# B&R Automation Studio project OpcUaSample410_BrbLibUa103 (part 21)

#### Action.st
```iecst
ACTION InitAirCond:
	// Logik
	pInstance.Act.eOperationMode := eAC_OPERATIONMODE_OFF;
	pInstance.Act.rTemperature := rAIR_COND_TEMP_OUTSIDE;
	pInstance.Act.nFanLevel := 0;
	pInstance.Set.rTemperature := 20.0;
	pInstance.Set.nFanLevel := 0;
END_ACTION

ACTION OperateAirCond:
	// Methode 'SetOperationMode'
	CASE pIntern.MethSetOperationMode.nStep OF
		0:
			// Prüfen, ob Methode von einem Client aufgerufen wurde
			pIntern.MethSetOperationMode.fbUaSrv_MethodOperate.Execute := 1;
			pIntern.MethSetOperationMode.fbUaSrv_MethodOperate.Action := UaMoa_CheckIsCalled;
			IF pIntern.MethSetOperationMode.fbUaSrv_MethodOperate.Done = 1 THEN
				pIntern.MethSetOperationMode.fbUaSrv_MethodOperate.Execute := 0;
				IF pIntern.MethSetOperationMode.fbUaSrv_MethodOperate.IsCalled = 1 THEN
					// Variablen der Eingans-Argumente sind besetzt -> Methode ausführen
					pIntern.MethSetOperationMode.nStep := 1;
				END_IF
			ELSIF pIntern.MethSetOperationMode.fbUaSrv_MethodOperate.Error = 1 THEN
				// Fehler, aber trotzdem weiter machen
				pIntern.MethSetOperationMode.fbUaSrv_MethodOperate.Execute := 0;
			END_IF

		1:
			// Ausführen der Methode
			IF pIntern.MethSetOperationMode.ArgsIn.eOperationMode >= eAC_OPERATIONMODE_OFF AND pIntern.MethSetOperationMode.ArgsIn.eOperationMode <= eAC_OPERATIONMODE_AUTO THEN
				pInstance.Act.eOperationMode := pIntern.MethSetOperationMode.ArgsIn.eOperationMode;
				pIntern.MethSetOperationMode.ArgsOut.eStatus := eAC_METH_STATUS_OK;
			ELSE
				pIntern.MethSetOperationMode.ArgsOut.eStatus := eAC_METH_STATUS_INVALID_OPMODE;
			END_IF
			pIntern.MethSetOperationMode.nStep := 2;

		2:
			// Rückmelden, dass Methode ausgeführt wurde. Zu diesem Zeitpunkt müssen die Ausgangs-Argumente besetzt sein und dürfen nicht mehr geändert werden
			pIntern.MethSetOperationMode.fbUaSrv_MethodOperate.Execute := 1;
			pIntern.MethSetOperationMode.fbUaSrv_MethodOperate.Action := UaMoa_Finished;
			IF pIntern.MethSetOperationMode.fbUaSrv_MethodOperate.Done = 1 THEN
				pIntern.MethSetOperationMode.fbUaSrv_MethodOperate.Execute := 0;
				pIntern.MethSetOperationMode.nStep := 0;
			ELSIF pIntern.MethSetOperationMode.fbUaSrv_MethodOperate.Error = 1 THEN
				// Fehler, aber trotzdem weiter machen
				pIntern.MethSetOperationMode.fbUaSrv_MethodOperate.Execute := 0;
				pIntern.MethSetOperationMode.nStep := 0;
			END_IF

	END_CASE
	pIntern.MethSetOperationMode.fbUaSrv_MethodOperate();

	// Begrenzung der SetTemp
	IF pInstance.Set.rTemperature < rAIR_COND_TEMP_MIN THEN
		pInstance.Set.rTemperature := rAIR_COND_TEMP_MIN;
	ELSIF pInstance.Set.rTemperature > rAIR_COND_TEMP_OUTSIDE THEN
		pInstance.Set.rTemperature := rAIR_COND_TEMP_OUTSIDE;
	END_IF
	// Berechnung der internen Werte (Abweichung in Prozent)
	pIntern.rDiff := pInstance.Act.rTemperature - pInstance.Set.rTemperature;
	pIntern.rDiffPercent := pIntern.rDiff / pInstance.Act.rTemperature * 100.0;
	// Steuern des Lüfters
	IF pInstance.Act.eOperationMode = eAC_OPERATIONMODE_OFF THEN
		// Lüfter ausschalten
		pInstance.Act.nFanLevel := 0;
	ELSIF pInstance.Act.eOperationMode = eAC_OPERATIONMODE_MANUAL THEN
		// Lüfter-Stufe aus manueller Vorgabe übernehmen
		IF pInstance.Set.nFanLevel > 5 THEN
			pInstance.Act.nFanLevel := 5;
		ELSE
			pInstance.Act.nFanLevel := pInstance.Set.nFanLevel;
		END_IF
	ELSIF pInstance.Act.eOperationMode = eAC_OPERATIONMODE_AUTO THEN
		// Lüfter-Stufe je nach Temperatur-Differenz setzen
		IF pIntern.rDiffPercent <= 0.0 THEN
			pInstance.Act.nFanLevel := 0;
		ELSIF pIntern.rDiffPercent <= 10.0 THEN
			pInstance.Act.nFanLevel := 1;
		ELSIF pIntern.rDiffPercent <= 15.0 THEN
			pInstance.Act.nFanLevel := 2;
		ELSIF pIntern.rDiffPercent <= 20.0 THEN
			pInstance.Act.nFanLevel := 3;
		ELSIF pIntern.rDiffPercent <= 25.0 THEN
			pInstance.Act.nFanLevel := 4;
		ELSE
			pInstance.Act.nFanLevel := 5;
		END_IF
	END_IF
	SimulateAirCond;

	// Event 'AirConditionOperationModeChanged'
	IF pInstance.Act.eOperationMode <> pIntern.EvntOperationModeChanged.eOldOperationMode THEN
		// Besetzen der Felder mit aktuellen Werten
		pIntern.EvntOperationModeChanged.Fields.OldOperationMode := pIntern.EvntOperationModeChanged.eOldOperationMode;
		pIntern.EvntOperationModeChanged.Fields.NewOperationMode := pInstance.Act.eOperationMode;
		sMessageText := 'Operation mode of air condition $'';
		brsstrcat(ADR(sMessageText), ADR(pInstance.sName));
		brsstrcat(ADR(sMessageText), ADR('$' has changed from $''));
		eOperationMode := pIntern.EvntOperationModeChanged.Fields.OldOperationMode;
		GetOperationModeText;
		brsstrcat(ADR(sMessageText), ADR(sOperationModeText));
		brsstrcat(ADR(sMessageText), ADR('$' to $''));
		eOperationMode := pIntern.EvntOperationModeChanged.Fields.NewOperationMode;
		GetOperationModeText;
		brsstrcat(ADR(sMessageText), ADR(sOperationModeText));
		brsstrcat(ADR(sMessageText), ADR('$' (ST).'));
		brsstrcpy(ADR(pIntern.EvntOperationModeChanged.Fields.Message.Text), ADR(sMessageText));
		// Event feuern
		pIntern.EvntOperationModeChanged.bFire := 1;
	END_IF
	pIntern.EvntOperationModeChanged.eOldOperationMode := pInstance.Act.eOperationMode;
	CASE pIntern.EvntOperationModeChanged.nStep OF
		0:
			// Ermitteln des Namespace-Index für Fremdmodell-Adressbereich am am B&R-Server
			pIntern.EvntOperationModeChanged.fbUaSrv_GetNamespaceIndex.Execute := 1;
			pIntern.EvntOperationModeChanged.fbUaSrv_GetNamespaceIndex.NamespaceUri := 'http://br-automation.com/AirCondModel/';
			IF pIntern.EvntOperationModeChanged.fbUaSrv_GetNamespaceIndex.Done = 1 THEN
				pIntern.EvntOperationModeChanged.fbUaSrv_GetNamespaceIndex.Execute := 0;
				pIntern.EvntOperationModeChanged.nNamespaceIndexAirCond := pIntern.EvntOperationModeChanged.fbUaSrv_GetNamespaceIndex.NamespaceIndex;
				brsitoa(pIntern.EvntOperationModeChanged.nNamespaceIndexAirCond, ADR(pIntern.EvntOperationModeChanged.sNamespaceIndexAirCond));
				pIntern.EvntOperationModeChanged.nStep := pIntern.EvntOperationModeChanged.nStep + 1;
			ELSIF pIntern.EvntOperationModeChanged.fbUaSrv_GetNamespaceIndex.Error = 1 THEN
				// Fehler
				pIntern.EvntOperationModeChanged.fbUaSrv_GetNamespaceIndex.Execute := 0;
			END_IF

		1:
			// Initialisierung zum Feuern des Events
			// Event-Typ
			pIntern.EvntOperationModeChanged.fbUaSrv_FireEvent.EventType.NamespaceIndex := pIntern.EvntOperationModeChanged.nNamespaceIndexAirCond;
			pIntern.EvntOperationModeChanged.fbUaSrv_FireEvent.EventType.IdentifierType := UAIdentifierType_Numeric;
			pIntern.EvntOperationModeChanged.fbUaSrv_FireEvent.EventType.Identifier := '1002'; // = AirConditionOperationModeChanged
			// Event-Felder
			nFieldIndex := 0;
			// SourceNode
			pIntern.EvntOperationModeChanged.Fields.FieldCfg[nFieldIndex].BrowsePath := '/SourceNode';
			sVarNameTotal := pIntern.EvntOperationModeChanged.sEventFieldsBaseVarName;
			brsstrcat(ADR(sVarNameTotal), ADR('.SourceNode'));
			pIntern.EvntOperationModeChanged.Fields.FieldCfg[nFieldIndex].Variable := sVarNameTotal;
			pIntern.EvntOperationModeChanged.Fields.SourceNode.NamespaceIndex := pIntern.EvntOperationModeChanged.nNamespaceIndexAirCond;
			pIntern.EvntOperationModeChanged.Fields.SourceNode.IdentifierType := UAIdentifierType_Numeric;
			pIntern.EvntOperationModeChanged.Fields.SourceNode.Identifier := pIntern.EvntOperationModeChanged.sEventFieldSourceNode;
			// Message
			nFieldIndex := nFieldIndex + 1;
			pIntern.EvntOperationModeChanged.Fields.FieldCfg[nFieldIndex].BrowsePath := '/Message';
			sVarNameTotal := pIntern.EvntOperationModeChanged.sEventFieldsBaseVarName;
			brsstrcat(ADR(sVarNameTotal), ADR('.Message'));
			pIntern.EvntOperationModeChanged.Fields.FieldCfg[nFieldIndex].Variable := sVarNameTotal;
			pIntern.EvntOperationModeChanged.Fields.Message.Text := 'Operation mode has changed.';
			// OldOperationMode
			nFieldIndex := nFieldIndex + 1;
			sFieldNameTotal := '/';
			brsstrcat(ADR(sFieldNameTotal), ADR(pIntern.EvntOperationModeChanged.sNamespaceIndexAirCond));
			brsstrcat(ADR(sFieldNameTotal), ADR(':OldOperationMode'));
			pIntern.EvntOperationModeChanged.Fields.FieldCfg[nFieldIndex].BrowsePath := sFieldNameTotal;
			sVarNameTotal := pIntern.EvntOperationModeChanged.sEventFieldsBaseVarName;
			brsstrcat(ADR(sVarNameTotal), ADR('.OldOperationMode'));
			pIntern.EvntOperationModeChanged.Fields.FieldCfg[nFieldIndex].Variable := sVarNameTotal;
			// NewOperationMode
			nFieldIndex := nFieldIndex + 1;
			sFieldNameTotal := '/';
			brsstrcat(ADR(sFieldNameTotal), ADR(pIntern.EvntOperationModeChanged.sNamespaceIndexAirCond));
			brsstrcat(ADR(sFieldNameTotal), ADR(':NewOperationMode'));
			pIntern.EvntOperationModeChanged.Fields.FieldCfg[nFieldIndex].BrowsePath := sFieldNameTotal;
			sVarNameTotal := pIntern.EvntOperationModeChanged.sEventFieldsBaseVarName;
			brsstrcat(ADR(sVarNameTotal), ADR('.NewOperationMode'));
			pIntern.EvntOperationModeChanged.Fields.FieldCfg[nFieldIndex].Variable := sVarNameTotal;
			// Statische Funktionsblock-Eingänge
			pIntern.EvntOperationModeChanged.fbUaSrv_FireEvent.EventFieldCount := nFieldIndex+1;
			pIntern.EvntOperationModeChanged.nStep := pIntern.EvntOperationModeChanged.nStep + 1;

		2:
			// Prüfen, ob Event gefeuert werden muss
			IF pIntern.EvntOperationModeChanged.bFire = 1 THEN
				pIntern.EvntOperationModeChanged.bFire := 0;
				pIntern.EvntOperationModeChanged.nStep := pIntern.EvntOperationModeChanged.nStep + 1;
			END_IF

		3:
			// Event feuern
			pIntern.EvntOperationModeChanged.fbUaSrv_FireEvent.Execute := 1;
			IF pIntern.EvntOperationModeChanged.fbUaSrv_FireEvent.Done = 1 THEN
				pIntern.EvntOperationModeChanged.fbUaSrv_FireEvent.Execute := 0;
				pIntern.EvntOperationModeChanged.nStep := pIntern.EvntOperationModeChanged.nStep - 1;
			ELSIF pIntern.EvntOperationModeChanged.fbUaSrv_FireEvent.Error = 1 THEN
				// Fehler
			END_IF

	END_CASE
	pIntern.EvntOperationModeChanged.fbUaSrv_GetNamespaceIndex();
	pIntern.EvntOperationModeChanged.fbUaSrv_FireEvent(EventFields := pIntern.EvntOperationModeChanged.Fields.FieldCfg[0]);

END_ACTION

ACTION SimulateAirCond:
	// Stetiges Angleichen an die Aussentemperatur
	pInstance.Act.rTemperature := pInstance.Act.rTemperature + 0.0005;
	IF pInstance.Act.rTemperature > rAIR_COND_TEMP_OUTSIDE THEN
		pInstance.Act.rTemperature := rAIR_COND_TEMP_OUTSIDE;
	END_IF
	// Kühlen
	IF pInstance.Act.eOperationMode <> eAC_OPERATIONMODE_OFF THEN
		// Je nach Lüfter-Stufe kühlt die ActTemp runter
		pIntern.rCoolStepTemp := pInstance.Act.nFanLevel * 0.005;
		pInstance.Act.rTemperature := pInstance.Act.rTemperature - pIntern.rCoolStepTemp;
	END_IF
	// Physikalische Begrenzung der ActTemp
	IF pInstance.Act.rTemperature < rAIR_COND_TEMP_MIN THEN
		pInstance.Act.rTemperature := rAIR_COND_TEMP_MIN;
	END_IF
END_ACTION

ACTION GetOperationModeText:
	IF eOperationMode = eAC_OPERATIONMODE_OFF THEN
		sOperationModeText := 'Off';
	ELSIF eOperationMode = eAC_OPERATIONMODE_MANUAL THEN
		sOperationModeText := 'Manual';
	ELSIF eOperationMode = eAC_OPERATIONMODE_AUTO THEN
		sOperationModeText := 'Automatic';
	ELSE
		sOperationModeText := 'Unknown';
	END_IF
END_ACTION
```

### ReadMe.txt
```
Hier wird die Konfiguration von Publisher/Subscriber gezeigt.

Allgemeines zu PubSub
	PubSub ist eine alternative OpcUa-Kommunikation zu einer Client-Server-Verbindung.
	Bei PubSub ist es im Gegensatz zu Client/Server nicht notwendig, eine explizite Verbindung aufzubauen. Der Publisher
	schickt die Daten autark durch ein Udp-Multicast-Telegramm ins Netzwerk. Dieses	Telegramm kann dann von einem oder
	mehreren Subscribern empfangen und ausgewertet werden. Der Publisher weiss nicht, ob und welche Subscriber zuhören.
	Eine B&R-Sps kann Publisher sein (und mehrere Datenblöcke in verschiedenen Intervallen publishen) und gleichzeitig
	Subscriber auf mehrere andere Publisher enthalten. Sie kann sich nur nicht auf einen Datenblock des eigenen Publishers
	abonnieren (Hintergrund siehe 'Zu diesem Beispiel' unten).

	Theoretisch muss ein Publisher oder ein Subscriber nicht gleichzeitig ein Server oder Client sein. Beide Kommunkationsarten
	haben lt. Spezifikation nichts miteinander zu tun.
	Praktisch ist es aber oft so, dass ein Publisher Knoten aus einem Adressraum veröffentlicht, der bequemerweise von einem
	Server bereitgestellt wird. Auch ein Subscriber benötigt einen Adressraum, auf dessen Knoten die empfangenen Daten kopiert
	werden können. Eine B&R-Sps braucht deshalb eine Adressraum-Konfiguration und auch das OpcUa-System muss in der System-
	Konfiguration aktiviert sein.

	PubSub wird oft zusammen mit TSN (TimeSensitiveNetwork, also echtzeitfähiges Ethernet) genannt. Tatsächlich wird PubSub
	von OpcUa-TSN verwendet. Trotzdem kann PubSub auch autaurk in nicht echtzeitfähigen Ethernet-Netzwerken eingesetzt
	werden. Dies ist hier der Fall, da TSN noch nicht veröffentlicht ist. Deshalb müssen auch die Parameter unter 'Activate VLAN'
	in der PubSub-Konfiguration noch nicht gesetzt werden (sie sind später für TSN wichtig).

	Laut Spezifikation hängt der Aufbau eines Publisher-Multicast-Telegramms (einer sogenannten NetworkMessage) von sehr
	vielen Optionen ab. Viele Parameter	werden nur optional im Telegramm mitgesendet. Es gibt auch einige spezifizierte
	Formate, sogenannte 'HeaderLayouts', welche den Aufbau zu großen Teilen festlegen. So kann die sonst sehr aufwändige
	Konfiguration stark vereinfacht	ausfallen. B&R nutzt das HeaderLayout 'UADP-Periodic-Fixed', mit dem viele Parameter
	fix gesetzt sind und so die	Konfiguration überschaubar macht.
	Es gibt auch einige Einschränkungen, welche in der AS-Hilfe genauer beschrieben sind:
		-Nur skalare Werte und 1-dimensionale Arrays
		-Keine Strukturen, Enumerationen, Pointer, Konstanten
		-Noch keine Security (Verschlüsselung)
		-Der Publisher wird nicht synchron zu den Taskklassen ausgeführt. Somit ist eine Konsistenz der Daten zueinander, auch
			wenn sie in einem DataSet sind, nicht gewährleistet. Diese Funktionalität wird erst durch TSN abgebildet werden
			können.

Zu diesem Beispiel
	Leider kann in einer ArSim (Sps-Simulation auf einem PC), wie sie für dieses Beispiel-Projekt verwendet wird, keine
	funktionierende PubSub-Verbindung gezeigt werden. Dafür gibt es mehrere Gründe:
		1. Eine Sps kann sich nicht selber zuhören, also auf den eigenen Publisher subscriben.
				Grund: Ethernet-Sockets sind auf der Sps so eingestellt, dass sie ihre gesendeteten Telegramme nicht gleichzeitig
				auch empfangen (auch nicht, wenn es Multicast-Telegramme sind). Dies hat performance-technische Gründe:
				Müsste ein Socket auch die selber gesendeten Telegramme empfangen und auswerten, würde dies die Hardware zu sehr
				durch Interrupts belasten.
		2. Eine ArSim hat normalerweise (wie hier auch) eine virtuelle Ethernet-Verbindung über die Adresse 127.0.0.1.
				Aufgrund des virtuellen Netzwerkes werden keine Telegramme vom Publisher veröffentlicht.

	Aus diesem Grund kann hier nur die exemplarische Konfiguration gezeigt werden. Würde dieses Beispiel auf zwei Hardware-
	Sps angepasst, so würde die Kommunikation funktionieren.

	Es gibt zumindest einen Trick, wie die Publisher-Multicast-Telegramme einer ArSim in ein äußeres Netzwerk des PC's gebracht
	werden können: Die Ip-Adresse der einzigen ArSim-Ethernet-Schnittstelle IF3, welche normalerweise auf 127.0.0.1 eingestellt
	ist, muss auf die Ip-Adresse des PC's zu dem Netzwerk eingestellt werden. Dann werden die Telegramme über Windows automatisch
	an diese Ethernet-Schnittstelle und somit in das Netzwerk geschickt. Sie können dann sogar mit Wireshark aufgezeichnet
	oder von einem Subscriber im Netzwerk empfangen werden. Leider funktioniert dies in Windows nur in diese Richtung. Von Windows
	empfangene Telegramme werden nicht auf die ArSim	weitergeleitet und können deshalb auch nicht von einem ArSim-Subscriber
	empfangen werden.
	Hinweis: Trotz dieses Tricks kann eine ArSim sich nicht selber zuhören (siehe oben).

	Eine PubSub-Configuration kann jeweils einen Publisher (in den WriterGrops) und einen Subscriber (in den ReaderGroups)
	enthalten. In diesem Beispiel sind sie der Übersichtlichkeit halber aber auf zwei separate PubSub-Konfigurationen
	('ExamplePublisher' und 'ExampleSubscriber') aufgeteilt.
```

### Package Logical/Tasks/PubSub/Publisher - Export der Publisher-Konfiguration

### ReadMe.txt
```
Hier wird die Konfiguration des Publishers erklärt.

	Die Konfiguration ist in der Datei 'UaPubSub.uaPubSub' unter 'ConfigurationView/ArSim/PC/Connectivity/OpcUA' enthalten.
	Hier können theoretisch beliebig viele Publisher konfiguriert werden.
	Achtung: Einige der Parameter werden nur angezeigt, wenn die erweiterte Parameter-Ansicht in der Symbol-Leiste angehakt ist!

	In diesem Beispiel ist ein Publisher konfiguriert, der zwei Datenblöcke in unterschiedlichen Intervallen sendet.
	Hierarchischer Aufbau und wichtige Parameter:
		+	ExamplePublisher									Ist gleichzeitig der Name der Publisher-Konfiguration. Dient nur der Unterscheidung
		|																			zu anderen Elementen. Es kann beliebig viele Konfigurationen geben.
		+-	Publisher ID										Dieser Parameter ermöglicht einem Subscriber, Daten eines bestimmten Publishers zu
		|																			abonnieren. Dieser Parameter gilt nur für die WriterGroups einer Publisher-
		|																			Konfiguration.
		+-	Network interface								Auswahl der Ethernet-Schnittstelle, an der gesendet wird.
		+-+	Address
		|	+-	IP address										Angabe der Multicast-Ip, an die gesendet wird. Sie muss zwischen 224.0.0.0 und
		|	|																		239.255.255.255 liegen. Dieser Bereich ist weltweit für Multicasts reserviert.
		|	|																		Diese Adresse ermöglicht einem Subscriber, bestimmte Publisher zu abonnieren.
		|	+-	Port number										Dieser Port ermöglicht einem Subscriber, bestimmte Publisher zu abonnieren.
		|																			Die Standard-Portnummer für OpcUa ist 4840, es kann jedoch auch eine andere
		|																			verwendet werden.
		+-+	WriterGroups										Es kann beliebig viele WriterGroups geben.
			+-	Name													Der Name dient nur der Unterscheidung zu anderen Elementen.
			+-	WriterGroup ID								Dieser Parameter ermöglicht einem Subscriber, bestimmte Daten eines Publishers zu
			|																		abonnieren.
		  +-	Publishing interval						In diesem Intervall in [ms] werden die unterliegenden Daten versendet.
			|																		Hier sollte bewusst eine Zeit gewählt werden, die ausreicht. Ein zu kleines
			|																		Intervall belastet unnötigerweise den Publisher, das Netzwerk und die Subscriber.
			|																		Das kleinste mögliche Intervall beträgt 10ms.
		  +-+	DataSetWriter									Es kann beliebig viele Writer innerhalb einer WriterGroup geben.
		  	+-	Name												Der Name dient nur der Unterscheidung zu anderen Elementen.
		  	+-	DataSetWriter ID						Dieser Parameter ermöglicht einem Subscriber, bestimmte Daten eines Publishers zu
				|																abonnieren. Ein B&R Subscriber wertet sie nicht aus.
		  	+-+	PublishedDataSet						Es gibt nur 1 DataSet pro Writer.
		  		+-	Name											Der Name dient nur der Unterscheidung zu anderen Elementen.
		  		+-+	DataSet field							Es kann mehrere Fields innerhalb des DataSets geben.
						+-	DataSet field name			Der Name dient nur der Unterscheidung zu anderen Elementen.
						+-	DataSet field ID				Wird vom Editor automatisch erstellt und dient einer zukünftigen Funktionalität.
						+-	Source variable					Stellt die Quelle des Wertes dieses Fields dar. Sie wird als NodeId des Server-
																				Adressraums angegeben.
																				Achtung: Der Knoten muss im Server-Adressraums freigegeben sein. Dabei ist es
																				unwichtig, welche Rechte für welche Rolle vergeben sind.

		Der Name eines Elements sollte aussagekräftig gewählt werden (vor allem bei Fields), da die Konfiguration hier exportiert
		(siehe unten 'Export') und bei einem Subscriber importiert werden kann. Der Projektierer des Subscribers kann dann
		aufgrund der Namen die Bedeutung der Elemente erkennen.

		Hier noch Informationen zu bestimmten Parametern:
			WriterGroup/Message settings/GroupVersion
				Die GroupVersion wird bei Änderung relevanter Parameter automatisch neu gesetzt. Sie berechnet sich aus den Sekunden
				seit 01.01.2000 als Uint32. Sie wird im Telegramm mitgeschickt und dient manchen Subscribern als Hinweis, dass ihre
				Konfiguration nicht mehr der des Publishers entspricht. Ein B&R Subscriber wertet sie nicht aus.

			Field/FieldMetaData
				Diese Angaben können nicht per Hand verändert werden, weil sie automatisch bei Auswahl der Quelle gesetzt werden.

		Notwendigkeit von verschiedenen Elementen
			Eine eigene Konfiguration muss immer dann verwendet werden, wenn unterschiedliche Multicast-Ip oder Ports verwendet
				werden sowie wenn an verschiedenen Ethernet-Schnittstellen gesendet werden soll. In diesem Beispiel wird nur eine
				Publisher-Konfiguration verwendet.
			Eine eigene WriterGroup muss immer dann angelegt werden, wenn Daten in verschiedenen Intervallen gesendet werden
				sollen. In diesem Beispiel wird in zwei Intervallen gesendet (500ms und 1000ms), weshalb auch zwei WriterGroups
				angelegt sind.
			Jeder Writer wird durch eine eigene NetworkMessage (also ein eigenes Multicast-Telegramm) versendet. Die darin
				enthaltene DataSetWriterId ermöglicht dem Subscriber die Filterung der Messages, die für ihn interessant sind.
				Verschiedene Writer sind also dann notwendig, wenn bestimmte Daten nur von bestimmten Subscribern benötigt werden.
				In diesem Beispiel sind in der ersten WriterGroup exemplarisch zwei Writer angelegt.

			Achtung: Ein Writer kann nur so viele Fields enthalten, dass die komplette Message nicht mehr als 1400 Bytes benötigt!

		Tasks
			-Quelle der Field-Werte
				Für die zu publishenden Werte der Fields werden Variablen aus dem Task 'ServerData' verwendet, welche zyklisch
				hochzählen. Deshalb ist hier kein	eigener Task notwendig.
				Hinweis: Es könnten auch globale Variablen verwendet werden. Es ist nur wichtig, dass die Variablen im Server-Adressraum
				freigegeben sind.
			-PubDiag
				Dieser Task enthält die Aufrufe zum Ermitteln der Publisher-Diagnose-Zähler (siehe unten). Da hier nur
				einfache Funktionsaufrufe benötigt werden, gibt es den Task nur in ANSI-C, nicht in StructuredText.

		Diagnose
			Der Publisher kann optional durch Zähler diagnostiziert werden (siehe Task 'PubDiag'), die über Funktionen der
			System-Bibliothek 'ArPubSubD' ermittelt werden. Sie zählen jeweils die gesendeten Messages (Telegramme) und DataSets,
			wobei immer die Gesamtanzahl und die Anzahl, bei denen Fehler aufgetreten sind, mitgezählt werden.
			Hinweis: Beim Hochlauf des Systems können immer ein paar Fehler gezählt werden.
			Treten im zyklischen Betrieb immer noch Fehler auf, sollte die Konfigurationen auf Parametrier-Fehler untersucht werden.
			Achtung: Bei einer ArSim mit Ip 127.0.0.1 werden keine Telegramme vom Publisher veröffentlicht (siehe
			PubSub/ReadMe.txt). Deshalb zählen die Diagnose-Zähler in diesem Beispiel nicht hoch.

		Export
			Durch den Kontext-Menü-Punkt 'Export all published datatsets for all connections to *.uabinary' können die gesamten
			Konfigurationen exportiert werden (es werden immer alle Publisher-Konfigurationen exportiert). Dieses Datei-Format ist
			durch die Opc-Foundation standardisiert und kann demnach zum Austausch mit Subscribern verwendet werden.
			Achtung: Der Kontext-Menü-Punkt ist nur dann sichtbar, wenn die PubSub-Konfiguration angewählt ist!
			Wenn ein Subscriber den Import dieses Formats erlaubt (wie z.B. das Automation Studio oder RnCommTest), kann auf
			diese Weise die	Konfiguration des Subscribers sehr stark vereinfacht werden.
			In diesem Beispiel ist die exportierte Datei mit dem Namen 'OpcUaSample49_PublisherExport.uabinary' vorhanden.

		Hinweise zu Strings
			Leider sind in der momentanen AS4.9 und der zugehörigen AR A4.90 noch einige Unzulänglichkeiten in Bezug auf den
			Datentyp STRING vorhanden:
				1. Zu publishende Strings oder String-Arrays dürfen nicht mit Konstanten, sondern nur mit Literalen (fixen Zahlen)
						deklariert sein.
				2. Änderung einer String-Deklaration bewirkt nicht automatisch eine Anpassung in der Publisher-Konfiguration.
			Diese Dinge werden wahrscheinlich in einer der nächsten Versionen behoben werden.
```

- OpcUaSample49_PublisherExport.uabinary (binary file, 2356 bytes)
### Program Logical/Tasks/PubSub/Publisher/PubDiag (ANSIC) - Publisher-Diagnose

#### PubDiag.c - Init, cyclic, exit code
```c
#include <bur/plctypes.h>

#ifdef _DEFAULT_INCLUDES
	#include <AsDefault.h>
#endif

// NOLINTBEGIN(readability-*, bugprone-easily-swappable-parameters, bugprone-branch-clone, clang-diagnostic-invalid-utf8, clang-diagnostic-invalid-source-encoding, clang-diagnostic-pointer-arith, clang-diagnostic-strict-prototypes, clang-diagnostic-shadow, clang-diagnostic-bad-function-cast, clang-analyzer-security.insecureAPI.*, hicpp-uppercase-literal-suffix, hicpp-function-size, cppcoreguidelines-*, performance-*)

void _INIT ProgramInit(void)
{

}

void _CYCLIC ProgramCyclic(void)
{
	// Diagnose-Zähler der gesendeten Messages
	PublisherDiagData.UdpMessage.nTotal = ArPubSubDGetUdpMsgSendTotal();
	PublisherDiagData.UdpMessage.nError = ArPubSubDGetUdpMsgSendError();
	// Diagnose-Zähler der gesendeten DataSets
	PublisherDiagData.DataSet.nTotal = ArPubSubDGetDataSetSendTotal();
	PublisherDiagData.DataSet.nError = ArPubSubDGetDataSetSendError();
}

void _EXIT ProgramExit(void)
{

}

// NOLINTEND(readability-*, bugprone-easily-swappable-parameters, bugprone-branch-clone, clang-diagnostic-invalid-utf8, clang-diagnostic-invalid-source-encoding, clang-diagnostic-pointer-arith, clang-diagnostic-strict-prototypes, clang-diagnostic-shadow, clang-diagnostic-bad-function-cast, clang-analyzer-security.insecureAPI.*, hicpp-uppercase-literal-suffix, hicpp-function-size, cppcoreguidelines-*, performance-*)
```

#### PubDiag.var - Local variables
```iecst
VAR
	PublisherDiagData : PubSubDiagData_TYP;
END_VAR
```

### ReadMe.txt
```
Hier wird die Konfiguration des Subscribers erklärt.

	Die Konfiguration ist in der Datei 'UaPubSub.uaPubSub' unter 'ConfigurationView/ArSim/PC/Connectivity/OpcUA' enthalten.
	Hier können theoretisch beliebig viele Subscriber konfiguriert werden.
	Achtung: Einige der Parameter werden nur angezeigt, wenn die erweiterte Parameter-Ansicht in der Symbol-Leiste angehakt ist!

	In diesem Beispiel ist ein Subscriber konfiguriert, alle Daten des eigenen Publishers empfangen könnte.
	Hierarchischer Aufbau und wichtige Parameter:
		+	ExampleSubscriber									Ist gleichzeitig der Name der Subscriber-Konfiguration. Dient nur der Unterscheidung
		|																			zu anderen Elementen. Es kann beliebig viele Konfigurationen geben.
		+-	Publisher ID										Dieser Parameter gilt nur für die WriterGroups einer Publisher-Konfiguration, ist also
		|																			für diese Subscriber-Konfiguration nicht wichtig.
		+-	Network interface								Auswahl der Ethernet-Schnittstelle, an der gehorcht wird.
		+-+	Address
		|	+-	IP address										Angabe der Multicast-Ip, auf die gehorcht wird.
		|	+-	Port number										Angabe des Ports, auf den gehorcht wird.
		+-+	ReaderGroups										Es kann beliebig viele ReaderGroups geben.
		  +-+	DataSetReader									Es kann beliebig viele Reader innerhalb einer ReaderGroup geben.
		  	+-	Name												Der Name dient nur der Unterscheidung zu anderen Elementen.
				+-	Publisher ID								Dieser Parameter wird zur Filterung der empfangenen Messages herangezogen.
				+-	WriterGroup ID							Dieser Parameter wird zur Filterung der empfangenen Messages herangezogen.
		  	+-	DataSetWriter ID						Dieser Parameter dient der Unterscheidung der DataSets, wird aber bei B&R nicht zur Filterung herangezogen.
				+-+	Message settings
				| +-	Group version							Sollte der Group version der Publisher-Konfiguration entsprechen.
				| +-	Network message number		Momentan immer 1.
				| +-	DataSet offset						Dieser Parameter gibt die Stelle an, an welcher die Daten dieses Readers in der
				|																	Message beginnen. Das Ermitteln dieses Parameters hängt von sehr vielen Optionen
				|																	des Publishers ab und ist daher sehr komplex. Am Besten sollte er durch Import der
				|																	Publisher-Konfiguration besetzt werden. Dann ist er auf jeden Fall richtig.
		  	+-+	SubscribedDataSet						Es gibt nur 1 DataSet pro Writer.
		  		+-	Name											Der Name dient nur der Unterscheidung zu anderen Elementen.
		  		+-+	DataSet field							Es kann mehrere Fields innerhalb des DataSets geben.
						+-	DataSet field name			Der Name dient nur der Unterscheidung zu anderen Elementen.
						+-	DataSet field ID				Dient einer zukünftigen Funktionalität.
						+-	Target variable					Gibt den Knoten im Adressraum an, auf den ein empfangener Wert geschrieben wird. Der
																				Datentyp des Knotens muss selbstverständlich zum Datentyp des Fields passen.
																				Achtung: Der Knoten muss im Server-Adressraums freigegeben sein. Dabei ist es
																				unwichtig, welche Rechte für welche Rolle vergeben sind.

		Hier noch Informationen zu bestimmten Parametern:
			Field/FieldMetaData
				Diese Angaben können nicht per Hand verändert werden, weil sie automatisch bei Auswahl des Targets gesetzt werden.

		Notwendigkeit von verschiedenen Elementen
			Eine eigene Konfiguration muss immer dann verwendet werden, wenn unterschiedliche Multicast-Ip oder Ports verwendet
				werden sowie wenn an verschiedenen Ethernet-Schnittstellen gehorcht werden soll. Aus diesem Grund wird in diesem
				Beispiel nur eine Subscriber-Konfiguration verwendet.
			Alle anderen Elemente müssen aus dem Publisher übernommen werden.

		Filterung von Messages
			Theoretisch können sehr viele Multicast-Telegramme von verschiedenen Publishern an der Sps eintreffen.
			Durch die Parameter der Subscriber-Konfiguration wird die Filterung der uninteressanten Messages vorgenommen. Diese
			wird in zwei Stufen durchgeführt:
				1. Die Firmware der Ethernet-Schnittstelle filtert auf die generellen Parameter, also auf Network-Interface,
						Multicast-Ip-Adresse und Port. Nur Telegramme, die diesen Parametern entsprechen, werden an das Betriebssystem
						weitergeleitet.
				2. Das Betriebssystem filtert auf alle unterliegenden Parameter von ReaderGroups und Reader, also auf
						PublisherId und WriterGroupId. Nur wenn dieser Filter passiert wurde, werden die enthaltenen
						DataSets ausgewertet und deren Werte übernommen.
			Daraus ergibt sich logischerweise: Wenn auch nur ein Parameter nicht mit den im gewünschten Publisher parametrierten
			Wert übereinstimmt, werden die Werte nicht übernommen! Es empfiehlt sich daher, die Konfiguration des Subscribers am
			Besten über die Import-Funktion zu machen (siehe 'Import' unten).

		Tasks
			-Subscriber
				Dieser Task enthält keinen Code, sondern stellt nur die Variablen zur Verfügung, auf welche die empfangenen Werte
				kopiert werden.
				Hinweis: Es könnten auch globale Variablen verwendet werden. Es ist nur wichtig, dass die Variablen im Server-Adressraum
				freigegeben sind.
			-SubDiag
				Dieser Task enthält die Aufrufe zum Ermitteln der Subscriber-Diagnose-Zähler (siehe) unten. Da hier nur
				einfache Funktionsaufrufe benötigt werden, gibt es den Task nur in ANSI-C, nicht in StructuredText.

		Diagnose
			Der Subscriber kann optional durch Zähler diagnostiziert werden (siehe Task 'SubDiag'), die über Funktionen der
			System-Bibliothek 'ArPubSubD' ermittelt werden. Sie zählen jeweils die empfangenen Messages (Telegramme) und DataSets,
			wobei immer die Gesamtanzahl und die Anzahl, bei denen Fehler aufgetreten sind, mitgezählt werden.
			Hinweis: Beim Hochlauf des Systems können immer ein paar Fehler gezählt werden.
			Treten im zyklischen Betrieb immer noch Fehler auf, sollte die Konfigurationen auf Parametrier-Fehler untersucht werden.
			Da die Diagnose im Betriebsystem stattfindet, umfasst sie auch nur Telegramme, welche den 1. Filter-Level (siehe oben)
			passiert haben.
			Achtung: Bei einer ArSim mit Ip 127.0.0.1 werden keine Telegramme vom Publisher veröffentlicht (siehe
			PubSub/ReadMe.txt) und vom Subscriber auch nicht empfangen. Deshalb zählen die Diagnose-Zähler in diesem Beispiel nicht
			hoch.

		Import
			Durch den Kontext-Menü-Punkt 'Import datatsets from *.uabinary' können die Konfigurationen eines Publishers importiert
			werden (es werden immer alle DataSets importiert; nicht benötigte können einfach wieder gelöscht werden).
			Achtung: Der Kontext-Menü-Punkt ist nur dann sichtbar, wenn der Knoten 'ReaderGroups' einer PubSub-Konfiguration
			angewählt ist!
			Generell ist diese Art der Konfiguration empfohlen, da sie Fehler ausschließt. Außerdem gibt es Parameter, die nicht
			so einfach zu ermitteln sind (z.B. DataSetOffset). Diese sind aber im Import enthalten und werden somit automatisch
			richtig gesetzt.
```

### Program Logical/Tasks/PubSub/Subscriber/Subscriber (ANSIC) - Subscriber-Variablen

#### Subscriber.c - Init, cyclic, exit code
```c
#include <bur/plctypes.h>

#ifdef _DEFAULT_INCLUDES
	#include <AsDefault.h>
#endif

// NOLINTBEGIN(readability-*, bugprone-easily-swappable-parameters, bugprone-branch-clone, clang-diagnostic-invalid-utf8, clang-diagnostic-invalid-source-encoding, clang-diagnostic-pointer-arith, clang-diagnostic-strict-prototypes, clang-diagnostic-shadow, clang-diagnostic-bad-function-cast, clang-analyzer-security.insecureAPI.*, hicpp-uppercase-literal-suffix, hicpp-function-size, cppcoreguidelines-*, performance-*)

void _INIT ProgramInit(void)
{
	// Variable verwenden, damit sie zumindest einmal im Code vorkommt und nicht vom Kompiler wegoptimiert wird
	brsmemset((UDINT)&SubscribedData, 0, sizeof(SubscribedData));
}

void _CYCLIC ProgramCyclic(void)
{
	// Dieser Task enthält keinen Code, sondern nur die Variablen-Deklaration zur Aufnahme der empfangenen Werte.
}

void _EXIT ProgramExit(void)
{

}

// NOLINTEND(readability-*, bugprone-easily-swappable-parameters, bugprone-branch-clone, clang-diagnostic-invalid-utf8, clang-diagnostic-invalid-source-encoding, clang-diagnostic-pointer-arith, clang-diagnostic-strict-prototypes, clang-diagnostic-shadow, clang-diagnostic-bad-function-cast, clang-analyzer-security.insecureAPI.*, hicpp-uppercase-literal-suffix, hicpp-function-size, cppcoreguidelines-*, performance-*)
```

#### Subscriber.typ - Local data types
```iecst
TYPE
	SubscribedData_TYP : 	STRUCT
		nUsint : USINT;
		nUint : UINT;
		nSint : SINT;
		nInt : INT;
		anInt : ARRAY[0..4]OF INT; (*INT[0..nOPCUA_ARRAY_INDEX_MAX]*)
	END_STRUCT;
END_TYPE
```

#### Subscriber.var - Local variables
```iecst
VAR
	SubscribedData : SubscribedData_TYP;
END_VAR
```

### Program Logical/Tasks/PubSub/Subscriber/SubDiag (ANSIC) - Subscriber-Diagnose

#### SubDiag.c - Init, cyclic, exit code
```c
#include <bur/plctypes.h>

#ifdef _DEFAULT_INCLUDES
	#include <AsDefault.h>
#endif

// NOLINTBEGIN(readability-*, bugprone-easily-swappable-parameters, bugprone-branch-clone, clang-diagnostic-invalid-utf8, clang-diagnostic-invalid-source-encoding, clang-diagnostic-pointer-arith, clang-diagnostic-strict-prototypes, clang-diagnostic-shadow, clang-diagnostic-bad-function-cast, clang-analyzer-security.insecureAPI.*, hicpp-uppercase-literal-suffix, hicpp-function-size, cppcoreguidelines-*, performance-*)

void _INIT ProgramInit(void)
{

}

void _CYCLIC ProgramCyclic(void)
{
	// Diagnose-Zähler der empfangenen Messages
	SubscriberDiagData.UdpMessage.nTotal = ArPubSubDGetUdpMsgReceiveTotal();
	SubscriberDiagData.UdpMessage.nError = ArPubSubDGetUdpMsgReceiveError();
	// Diagnose-Zähler der empfangenen DataSets
	SubscriberDiagData.DataSet.nTotal = ArPubSubDGetDataSetReceiveTotal();
	SubscriberDiagData.DataSet.nError = ArPubSubDGetDataSetReceiveError();
}

void _EXIT ProgramExit(void)
{

}

// NOLINTEND(readability-*, bugprone-easily-swappable-parameters, bugprone-branch-clone, clang-diagnostic-invalid-utf8, clang-diagnostic-invalid-source-encoding, clang-diagnostic-pointer-arith, clang-diagnostic-strict-prototypes, clang-diagnostic-shadow, clang-diagnostic-bad-function-cast, clang-analyzer-security.insecureAPI.*, hicpp-uppercase-literal-suffix, hicpp-function-size, cppcoreguidelines-*, performance-*)
```

#### SubDiag.var - Local variables
```iecst
VAR
	SubscriberDiagData : PubSubDiagData_TYP;
END_VAR
```

Listed in the project but not available here: Logical/UnitTests/UtBrbUaTemplate/testSuite.c, Logical/UnitTests/UtBrbLibUa/UtBrbUaStatus/testSuite.c, Logical/UnitTests/UtBrbLibUa/UtBrbUaNodes/testSuite.c, Logical/UnitTests/UtBrbLibUa/UtBrbUaAttributes/testSuite.c, Logical/UnitTests/UtBrbLibUa/UtBrbUaVariantValues/testSuite.c, Logical/UnitTests/UtBrbLibUa/UtBrbUaByteStrings/testSuite.c, Logical/UnitTests/UtBrbLibUa/UtBrbUaLocalizedTexts/testSuite.c, Logical/UnitTests/UtBrbLibUa/UtBrbUaQualifiedNames/testSuite.c, Logical/UnitTests/UtBrbLibUa/UtBrbUaTimeAndDate/testSuite.c, Logical/UnitTests/UtBrbLibUa/UtBrbUaAdditional/testSuite.c, Logical/UnitTests/UtBrbLibUa/UtBrbUaClient/testSuite.c, Logical/UnitTests/UtBrbLibUa/UtBrbUaServer/testSuite.c, Logical/Tasks/Template/G_Template.typ, Logical/Tasks/Template/G_Template.var, Logical/Tasks/Template/TemplateC/TemplateC/TemplateC.typ, Logical/Tasks/Template/TemplateC/TemplateC/TemplateC.var, Logical/Tasks/Template/TemplateST/TemplateST/TemplateST.typ, Logical/Tasks/Template/TemplateST/TemplateST/TemplateST.var, Logical/Tasks/ServerData/G_ServerData.typ, Logical/Tasks/ServerDt64/G_ServerDt64.typ, Logical/Tasks/ServerDt64/G_ServerDt64.var, Logical/Tasks/ServerMethods/SrvMethC/SrvMethC/SrvMethC.typ, Logical/Tasks/ServerMethods/SrvMethC/SrvMethC/SrvMethC.var, Logical/Tasks/ServerEvents/SrvEvntST/SrvEvntST/Types.typ, Logical/Tasks/ServerEvents/SrvEvntST/SrvEvntST/Variables.var, Logical/Tasks/Clients/ClientST/ClientST/ClientST.typ, Logical/Tasks/OpcUaAny/G_OpcUaAny.typ, Logical/Tasks/OpcUaAny/G_OpcUaAny.var, Logical/Tasks/BrbUa/BrbUaClient/G_BrbUaClient.typ, Logical/Tasks/BrbUa/BrbUaClient/G_BrbUaClient.var, Logical/Tasks/BrbUa/BrbUaClient/BrbUaCltC/BrbUaCltC/BrbUaCltC.typ, Logical/Tasks/BrbUa/BrbUaClient/BrbUaCltST/BrbUaCltST/BrbUaCltST.typ, Logical/Tasks/BrbUa/BrbUaServer/G_BrbUaServer.typ, Logical/Tasks/BrbUa/BrbUaServer/G_BrbUaSerber.var, Logical/Tasks/BrbUa/BrbUaServer/BrbUaSrvC/BrbUaSrvC/BrbUaSrvC.typ, Logical/Tasks/BrbUa/BrbUaServer/BrbUaSrvST/BrbSrvDatST/BrbUaSrvST.typ, Logical/Tasks/UaCerts/UaCertsC/UaCertsC/UaCertsC.typ, Logical/Tasks/UaCerts/UaCertsC/UaCertsC/UaCertsC.var, Logical/Tasks/AirCond/AirCondC/AirCondC/AirCondC.typ, Logical/Tasks/AirCond/AirCondST/AirCondST/AirCondST.typ, Logical/Tasks/PubSub/Publisher/PubDiag/PubDiag.typ, Logical/Tasks/PubSub/Subscriber/SubDiag/SubDiag.typ
